{attribute addProperty BoxType "EK1100-0000-0018"}
{attribute addProperty Id "Beckhoff_EL33xxEK1122Beckhoff_EL33xxEK1122_B04A0A54162A_0001_EL3311_0000_0016EL3311_E1732F4B15419.25A_0002_EL3311_0000_0017EL3311_E1732F4B15419.25A_0003_EL3311_0000_0018EL3311_3C1AE90C11414.25A_0004_EL3311_0000_0019EL3311_3C1AE90C11414.25A_0005_EL3311_0000_0020EL3311_3C1AE90C11414.25A_0006_EL3311_0000_0021EL3311_3C1AE90C11414.25A_0007_EL3311_0000_0022EL3311_3C1AE90C11414.25A_0008_EL3311_0000_0023EL3311_3C1AE90C11414.25A_0009_EL3312_0000_0016EL3312_4A09AC1222628.25A_0010_EL3312_0000_0017EL3312_4A09AC1222628.25A_0011_EL3312_0000_0018EL3312_1AB44F6514618.25A_0012_EL3312_0000_0019EL3312_1AB44F6514618.25A_0013_EL3312_0000_0020EL3312_1AB44F6514618.25A_0014_EL3312_0000_0021EL3312_1AB44F6514618.25A_0015_EL3312_0000_0022EL3312_1AB44F6514618.25A_0016_EL3312_0000_0023EL3312_1AB44F6514618.25A_0017_EL3314_0000_0016EL3314_D4A7958637046.25A_0018_EL3314_0000_0017EL3314_D4A7958637046.25A_0019_EL3314_0000_0018EL3314_61F3DCF521026.25A_0020_EL3314_0000_0019EL3314_61F3DCF521026.25A_0021_EL3314_0000_0020EL3314_61F3DCF521026.25A_0022_EL3314_0000_0021EL3314_61F3DCF521026.25A_0023_EL3314_0000_0022EL3314_61F3DCF521026.25A_0024_EL3314_0000_0023EL3314_61F3DCF521026.25A_0025_EL3314_0000_0024EL3314_61F3DCF521026.25A_0026_EL3314_0002_0016EL3314_BFD3528727434.25A_0027_EL3314_0010_0016EL3314_FE14BA1D58272.75A_0028_EL3314_0010_0017EL3314_FE14BA1D58272.75A_0029_EL3314_0010_0018EL3314_FA2A45DB27434.25A_0030_EL3314_0010_0019EL3314_FA2A45DB27434.25A_0031_EL3314_0010_0020EL3314_AAA7BA7127434.25A_0032_EL3314_0010_0021EL3314_AAA7BA7127434.25A_0033_EL3314_0090_0016EL3314_A69716D721026.25A_0034_EL3314_0090_0017EL3314_A69716D721026.25A_0035_EL3318_0000_0016EL3318_1D97BE52954119.25A_0036_EL3318_0000_0017EL3318_1D97BE52954119.25A_0037_EL3318_0000_0018EL3318_1D97BE52954119.25A_0038_EL3318_0000_0019EL3318_1D97BE52954119.25A_0039_EL3318_0000_0020EL3318_1D97BE52954119.25A_0040_EL3318_0000_0021EL3318_1D97BE52954119.25A_0041_EL3318_0000_0022EL3318_1D97BE52954119.25A_0042_EL3351_0000_0016EL3351_952A9D2322628.25A_0043_EL3351_0000_0017EL3351_952A9D2322628.25A_0044_EL3351_0000_0018EL3351_952A9D2322628.25A_0045_EL3351_0000_0019EL3351_952A9D2322628.25A_0046_EL3351_0000_0020EL3351_952A9D2322628.25A_0047_EL3356_0000_0017EL3356_16C4FA1F14618.25A_0048_EL3356_0000_0018EL3356_16C4FA1F14618.25A_0049_EL3356_0000_0019EL3356_16C4FA1F14618.25A_0050_EL3356_0000_0020EL3356_16C4FA1F14618.25A_0051_EL3356_0000_0021EL3356_38C5F1FD14618.25A_0052_EL3356_0000_0022EL3356_38C5F1FD14618.25A_0053_EL3356_0000_0023EL3356_38C5F1FD14618.25A_0054_EL3356_0000_0024EL3356_38C5F1FD14618.25A_0055_EL3356_0000_0025EL3356_38C5F1FD14618.25A_0056_EL3356_0010_0017EL3356_84E6850014618.25A_0057_EL3356_0010_0018EL3356_84E6850014618.25A_0058_EL3356_0010_0019EL3356_84E6850014618.25A_0059_EL3356_0010_0020EL3356_84E6850014618.25A_0060_EL3356_0010_0021EL3356_AAE78EE214618.25A_0061_EL3356_0010_0022EL3356_AAE78EE214618.25A_0062_EL3356_0010_0023EL3356_AAE78EE214618.25A_0063_EL3356_0010_0024EL3356_AAE78EE214618.25A_0064_EL3356_0010_0025EL3356_AAE78EE214618.25A_0065_EL3356_0020_0025EL3356_AAE78EE214618.25A_0066_EL3356_0090_0025EL3356_AAE78EE214618.25"}
{attribute addProperty CRC "3092208952"}
{attribute addProperty SizeInBites "18228"}
{attribute addProperty SizeInBytes "2278.5"}
TYPE Beckhoff_EL33xx_B84F5D38 EXTENDS EK1100_179A0949 :
STRUCT
	{attribute addProperty Name "Beckhoff_EL33xxEK1122"}
	Beckhoff_EL33xxEK1122 : Beckhoff_EL33xxEK1122_B04A0A54;
	{attribute addProperty Name "A_0001_EL3311_0000_0016"}
	A_0001_EL3311_0000_0016 : EL3311_E1732F4B;
	{attribute addProperty Name "A_0002_EL3311_0000_0017"}
	A_0002_EL3311_0000_0017 : EL3311_E1732F4B;
	{attribute addProperty Name "A_0003_EL3311_0000_0018"}
	A_0003_EL3311_0000_0018 : EL3311_3C1AE90C;
	{attribute addProperty Name "A_0004_EL3311_0000_0019"}
	A_0004_EL3311_0000_0019 : EL3311_3C1AE90C;
	{attribute addProperty Name "A_0005_EL3311_0000_0020"}
	A_0005_EL3311_0000_0020 : EL3311_3C1AE90C;
	{attribute addProperty Name "A_0006_EL3311_0000_0021"}
	A_0006_EL3311_0000_0021 : EL3311_3C1AE90C;
	{attribute addProperty Name "A_0007_EL3311_0000_0022"}
	A_0007_EL3311_0000_0022 : EL3311_3C1AE90C;
	{attribute addProperty Name "A_0008_EL3311_0000_0023"}
	A_0008_EL3311_0000_0023 : EL3311_3C1AE90C;
	{attribute addProperty Name "A_0009_EL3312_0000_0016"}
	A_0009_EL3312_0000_0016 : EL3312_4A09AC12;
	{attribute addProperty Name "A_0010_EL3312_0000_0017"}
	A_0010_EL3312_0000_0017 : EL3312_4A09AC12;
	{attribute addProperty Name "A_0011_EL3312_0000_0018"}
	A_0011_EL3312_0000_0018 : EL3312_1AB44F65;
	{attribute addProperty Name "A_0012_EL3312_0000_0019"}
	A_0012_EL3312_0000_0019 : EL3312_1AB44F65;
	{attribute addProperty Name "A_0013_EL3312_0000_0020"}
	A_0013_EL3312_0000_0020 : EL3312_1AB44F65;
	{attribute addProperty Name "A_0014_EL3312_0000_0021"}
	A_0014_EL3312_0000_0021 : EL3312_1AB44F65;
	{attribute addProperty Name "A_0015_EL3312_0000_0022"}
	A_0015_EL3312_0000_0022 : EL3312_1AB44F65;
	{attribute addProperty Name "A_0016_EL3312_0000_0023"}
	A_0016_EL3312_0000_0023 : EL3312_1AB44F65;
	{attribute addProperty Name "A_0017_EL3314_0000_0016"}
	A_0017_EL3314_0000_0016 : EL3314_D4A79586;
	{attribute addProperty Name "A_0018_EL3314_0000_0017"}
	A_0018_EL3314_0000_0017 : EL3314_D4A79586;
	{attribute addProperty Name "A_0019_EL3314_0000_0018"}
	A_0019_EL3314_0000_0018 : EL3314_61F3DCF5;
	{attribute addProperty Name "A_0020_EL3314_0000_0019"}
	A_0020_EL3314_0000_0019 : EL3314_61F3DCF5;
	{attribute addProperty Name "A_0021_EL3314_0000_0020"}
	A_0021_EL3314_0000_0020 : EL3314_61F3DCF5;
	{attribute addProperty Name "A_0022_EL3314_0000_0021"}
	A_0022_EL3314_0000_0021 : EL3314_61F3DCF5;
	{attribute addProperty Name "A_0023_EL3314_0000_0022"}
	A_0023_EL3314_0000_0022 : EL3314_61F3DCF5;
	{attribute addProperty Name "A_0024_EL3314_0000_0023"}
	A_0024_EL3314_0000_0023 : EL3314_61F3DCF5;
	{attribute addProperty Name "A_0025_EL3314_0000_0024"}
	A_0025_EL3314_0000_0024 : EL3314_61F3DCF5;
	{attribute addProperty Name "A_0026_EL3314_0002_0016"}
	A_0026_EL3314_0002_0016 : EL3314_BFD35287;
	{attribute addProperty Name "A_0027_EL3314_0010_0016"}
	A_0027_EL3314_0010_0016 : EL3314_FE14BA1D;
	{attribute addProperty Name "A_0028_EL3314_0010_0017"}
	A_0028_EL3314_0010_0017 : EL3314_FE14BA1D;
	{attribute addProperty Name "A_0029_EL3314_0010_0018"}
	A_0029_EL3314_0010_0018 : EL3314_FA2A45DB;
	{attribute addProperty Name "A_0030_EL3314_0010_0019"}
	A_0030_EL3314_0010_0019 : EL3314_FA2A45DB;
	{attribute addProperty Name "A_0031_EL3314_0010_0020"}
	A_0031_EL3314_0010_0020 : EL3314_AAA7BA71;
	{attribute addProperty Name "A_0032_EL3314_0010_0021"}
	A_0032_EL3314_0010_0021 : EL3314_AAA7BA71;
	{attribute addProperty Name "A_0033_EL3314_0090_0016"}
	A_0033_EL3314_0090_0016 : EL3314_A69716D7;
	{attribute addProperty Name "A_0034_EL3314_0090_0017"}
	A_0034_EL3314_0090_0017 : EL3314_A69716D7;
	{attribute addProperty Name "A_0035_EL3318_0000_0016"}
	A_0035_EL3318_0000_0016 : EL3318_1D97BE52;
	{attribute addProperty Name "A_0036_EL3318_0000_0017"}
	A_0036_EL3318_0000_0017 : EL3318_1D97BE52;
	{attribute addProperty Name "A_0037_EL3318_0000_0018"}
	A_0037_EL3318_0000_0018 : EL3318_1D97BE52;
	{attribute addProperty Name "A_0038_EL3318_0000_0019"}
	A_0038_EL3318_0000_0019 : EL3318_1D97BE52;
	{attribute addProperty Name "A_0039_EL3318_0000_0020"}
	A_0039_EL3318_0000_0020 : EL3318_1D97BE52;
	{attribute addProperty Name "A_0040_EL3318_0000_0021"}
	A_0040_EL3318_0000_0021 : EL3318_1D97BE52;
	{attribute addProperty Name "A_0041_EL3318_0000_0022"}
	A_0041_EL3318_0000_0022 : EL3318_1D97BE52;
	{attribute addProperty Name "A_0042_EL3351_0000_0016"}
	A_0042_EL3351_0000_0016 : EL3351_952A9D23;
	{attribute addProperty Name "A_0043_EL3351_0000_0017"}
	A_0043_EL3351_0000_0017 : EL3351_952A9D23;
	{attribute addProperty Name "A_0044_EL3351_0000_0018"}
	A_0044_EL3351_0000_0018 : EL3351_952A9D23;
	{attribute addProperty Name "A_0045_EL3351_0000_0019"}
	A_0045_EL3351_0000_0019 : EL3351_952A9D23;
	{attribute addProperty Name "A_0046_EL3351_0000_0020"}
	A_0046_EL3351_0000_0020 : EL3351_952A9D23;
	{attribute addProperty Name "A_0047_EL3356_0000_0017"}
	A_0047_EL3356_0000_0017 : EL3356_16C4FA1F;
	{attribute addProperty Name "A_0048_EL3356_0000_0018"}
	A_0048_EL3356_0000_0018 : EL3356_16C4FA1F;
	{attribute addProperty Name "A_0049_EL3356_0000_0019"}
	A_0049_EL3356_0000_0019 : EL3356_16C4FA1F;
	{attribute addProperty Name "A_0050_EL3356_0000_0020"}
	A_0050_EL3356_0000_0020 : EL3356_16C4FA1F;
	{attribute addProperty Name "A_0051_EL3356_0000_0021"}
	A_0051_EL3356_0000_0021 : EL3356_38C5F1FD;
	{attribute addProperty Name "A_0052_EL3356_0000_0022"}
	A_0052_EL3356_0000_0022 : EL3356_38C5F1FD;
	{attribute addProperty Name "A_0053_EL3356_0000_0023"}
	A_0053_EL3356_0000_0023 : EL3356_38C5F1FD;
	{attribute addProperty Name "A_0054_EL3356_0000_0024"}
	A_0054_EL3356_0000_0024 : EL3356_38C5F1FD;
	{attribute addProperty Name "A_0055_EL3356_0000_0025"}
	A_0055_EL3356_0000_0025 : EL3356_38C5F1FD;
	{attribute addProperty Name "A_0056_EL3356_0010_0017"}
	A_0056_EL3356_0010_0017 : EL3356_84E68500;
	{attribute addProperty Name "A_0057_EL3356_0010_0018"}
	A_0057_EL3356_0010_0018 : EL3356_84E68500;
	{attribute addProperty Name "A_0058_EL3356_0010_0019"}
	A_0058_EL3356_0010_0019 : EL3356_84E68500;
	{attribute addProperty Name "A_0059_EL3356_0010_0020"}
	A_0059_EL3356_0010_0020 : EL3356_84E68500;
	{attribute addProperty Name "A_0060_EL3356_0010_0021"}
	A_0060_EL3356_0010_0021 : EL3356_AAE78EE2;
	{attribute addProperty Name "A_0061_EL3356_0010_0022"}
	A_0061_EL3356_0010_0022 : EL3356_AAE78EE2;
	{attribute addProperty Name "A_0062_EL3356_0010_0023"}
	A_0062_EL3356_0010_0023 : EL3356_AAE78EE2;
	{attribute addProperty Name "A_0063_EL3356_0010_0024"}
	A_0063_EL3356_0010_0024 : EL3356_AAE78EE2;
	{attribute addProperty Name "A_0064_EL3356_0010_0025"}
	A_0064_EL3356_0010_0025 : EL3356_AAE78EE2;
	{attribute addProperty Name "A_0065_EL3356_0020_0025"}
	A_0065_EL3356_0020_0025 : EL3356_AAE78EE2;
	{attribute addProperty Name "A_0066_EL3356_0090_0025"}
	A_0066_EL3356_0090_0025 : EL3356_AAE78EE2;
END_STRUCT
END_TYPE

(* stored: Version 1.2.0.0, ProductVersion 3.1.4024.9
   DUT Beckhoff_EL33xx_B84F5D38: Id {6681eb42-bb00-4c63-bc11-a271bb28bce0} *)
